{attribute 'linkalways'} 
{attribute 'no_explicit_call' := 'This FB is a CLASS and must be accessed using methods or properties'}
{attribute 'enable_dynamic_creation'}
FUNCTION_BLOCK FINAL SUB_LWORD EXTENDS Node
VAR
	in1 : _LWORD(0);
	in2 : _LWORD(0);
	out : _LWORD(0);
END_VAR

METHOD PUBLIC Clone : I_Node
VAR
	pNode : POINTER TO SUB_LWORD;
END_VAR
pNode := __NEW(SUB_LWORD);
Clone := pNode^;
END_METHOD

METHOD FB_init : BOOL
VAR_INPUT
	bInitRetains : BOOL; // if TRUE, the retain variables are initialized (warm start / cold start)
	bInCopyCode : BOOL;  // if TRUE, the instance afterwards gets moved into the copy code (online change)
END_VAR
AddInput('in1',THIS^.in1);
AddInput('in2',THIS^.in2);
AddOutput('out', THIS^.out);
END_METHOD

METHOD PROTECTED OnExecute
VAR
END_VAR
out.Value := in1.Value - in2.Value;
END_METHOD

END_FUNCTION_BLOCK

(* stored: Version 1.1.0.1, ProductVersion 3.1.4024.15
   POU SUB_LWORD: Id {df0bde0d-705b-46c2-a703-5a3bd4974b11}, SpecialFunc None
   Folder Constructor: Id {ba61df0e-3758-4e09-8a8c-1474f6c46927}
   Method Clone: Id {0409de18-5bc0-46c6-96fb-9f0035f468dd}
   Method FB_init: Id {2eddf3fc-e8ea-4be6-8cdb-707b5a1bbdd8}
   Method OnExecute: Id {26a0dfc9-2fa6-4160-8cfb-204facfb3261} *)
